Universal Robots PolyScope program: dev_test_1.urp

Program dev_test_1 (installation=default directory=/ursim/programs createdIn=5.22.2 lastSavedIn=5.22.2 robotSerialNumber=20195599999)
Calibrated DH parameters: a=[0, -0.425, -0.3922, 0, 0, 0]; d=[0.1625, 0, 0, 0.1333, 0.0997, 0.0996]; alpha=[1.570796, 0, 0, 1.570796, -1.570796, 0]; deltaTheta=[0, 0, 0, 0, 0, 0]
InitVariablesNode
Robot Program (runOnlyOnce=false)
  Script file /ursim/programs/scripts/home_position.script
    | # Define the joint angles for the home position, as taken from docs.
    | # This is the same as clicking "home position" on polyclops.
    | # Remember the array is [base, shoulder, elbow, wrist1, wrist2, wrist3]
    | # Degrees to rad conversion: value in degrees �� ��/180 = rad
    | # Why the negative if 90 �� ��/180 = 1.5708? We use negative becase UR defines forward for the shoulder as negative rotation.
    | # Negative angles just mean ���rotate clockwise��� around the joint���s axis (from the joint���s frame of reference).
    | # This is why the home pose has negative values for the shoulder and elbow.
    | 
    | home_joint_positions = [0, -1.5708, 0, -1.5708,  0, 0]
    | 
    | # Move the robot to the defined position, with acceleration as 'a' and velocity parameter as v
    | 
    | movej(home_joint_positions, a = 1.5, v = 0.5)
  Script file /ursim/programs/scripts/pickup_target_one.script
    | on_target_position = [0, -1.918888889, -2.79253, 0, 1.5708, 0]
    | 
    | # Move the robot to the definde position, with acceleration as 'a' and velocity parameter as 0.5
    | # movej equals move joints
    | movej(on_target_position, a=1.5, v=0.5)
  Script file /ursim/programs/scripts/execute_gripping_action.script
    | #Executes the gripping action
  Script file /ursim/programs/scripts/move_to_drop_position_one.script
    | current_pose = get_actual_tcp_pose()
    | 
    | target_pose = pose_add(current_pose, p[0, 0.20, 0, 0, 0, 0])
    | 
    | movel(target_pose, a=1.0, v=0.25)
    | 
    | target_pose = pose_add(current_pose, p[0.40, 0, 0, 0, 0, 0])
    | 
    | movel(target_pose, a=1.0, v=0.25)
    | 
    | target_pose = pose_add(current_pose, p[0, -0.20, 0, 0, 0, 0])
    | 
    | movel(target_pose, a=1.0, v=0.25)
